FUNCTION F_CreateDynTextDefaultS : ST_Text
VAR_INPUT
	sText	: STRING;
END_VAR
VAR
END_VAR

F_CreateDynTextDefaultS.wsNameId := TO_WSTRING(sText);
F_CreateDynTextDefaultS.wsName := F_CreateDynTextDefaultS.wsNameId;

END_FUNCTION

(* stored: Version 1.1.0.1, ProductVersion 3.1.4024.12
   POU F_CreateDynTextDefaultS: Id {cc597b3b-78a4-42d2-aad9-ed4e396eb5df}, SpecialFunc None *)
